(* Logix 5000 project; controller cal1632 1756-L62 rev 16.20; software revision 16.05; part 56 of 61 *)
(* tags used below, declared in another part *)
   abs_distance_to_move : REAL;   // Turret Absolute Distance to Move
   distance_to_move : REAL;   // Turret Distence to Move
   last_selected_position : REAL;   // Turret Last Selected Position
   p29_param_tension_hi_limit : REAL;   // Parameter Tension High Limit
   param_doff_position : REAL;
   param_pos_db : REAL;   // C: Turret Position Dead Band
   pb_jog_turret_rev : BOOL;   // HMI PB: Jog Turret Rev
   pos_hi_limit : REAL;   // Turret Position DB High Limit
   pos_hi_limit_temp : REAL;   // Turret Position High Limit Temp
   pos_lo_limit : REAL;   // Turret Position DB Low Limit
   pos_lo_limit_temp : REAL;   // Turret Position Low Limit Temp
   tmr_fwd_delay : TIMER;   // Turret Signal Dwell Timer
   tmr_ref_delay : TIMER;   // Turret Signal Dwell Timer
   turret_err_mod : REAL;   // Turret Shortest Path Error wrapped to 0..360
   turret_err_raw : REAL;   // Turret Shortest Path Raw error plus 540 offset
   turret_in_wda_run_position : BOOL;   // Turret In Winder A Run Position
   turret_in_wdb_run_position : BOOL;   // Turret In Winder B Run Position
   turret_index_active_last_scan : BOOL;   // Turret Index Active Last Scan
   turret_index_permissive : BOOL;   // Turret Index Permissive No Turret Drive Fault AND Neither Winder Requesting Run
   turret_request_reverse : BOOL;   // Turret Request Reverse Index
   turret_wa_pos_doff_request : BOOL;   // Turret Move to Winder A Doff Position Request
   turret_wa_pos_run_request : BOOL;   // Turret Move to Winder A Run Position
   turret_wb_pos_doff_request : BOOL;   // Turret Move to Winder B Doff Position Request
   turret_wb_pos_run_request : BOOL;   // Turret Move to Winder B Run Position
   wa_doff_pos : REAL;   // Turret Winder A Doff Position
   wb_doff_pos_tmp : REAL;   // Turret Temp Doff Position before MOD
   wb_doff_position : REAL;   // Turret Winder B Doff Position
   wb_run_position : REAL;   // Turret Winder B Run Position
   wb_run_position_tmp : REAL;   // Turret Temp Run Position before MOD
   FAULT : BOOL;
   HMI : BOOL;
   p01_param_tension_deviation : REAL;
   p01_recipe_active : recipe;
   p01r02_plc_scan_time_in_sec : REAL;
   p01r09_pb_global_reset : BOOL;
   p01r13_permissive_drives : BOOL;
   p01r13_state : DINT;
   p25_ao_selected_speed : REAL;
   p29_ai_wa_rpm : REAL;
   p29_ai_wb_rpm : REAL;
   p29_ai_wdr_dia_in : REAL;
   p29_ai_wdr_lc : REAL;
   p29_ao_wdr_turret_selected_speed : REAL;
   p29_di_wdr_a_core_size : BOOL;
   p29_di_wdr_a_reset_core : BOOL;
   p29_di_wdr_b_core_size : BOOL;
   p29_di_wdr_b_reset_core : BOOL;
   p29_di_wdr_index_fwd : BOOL;
   p29_di_wdr_turret : acs800_di_normal;
   p29_di_wt_motor : BOOL;
   p29_do_wdr_turret : acs800_do_normal;
   p29_param_fast_turret_speed : REAL;
   p29_param_slow_turret_speed : REAL;
   p29_param_wa_gear_ratio : REAL;
   p29_param_wb_gear_ratio : REAL;
   p29_winder_at_run_position : BOOL;
   p29r01 : routine;
   p29r09_mode_doff_auto : BOOL;   // Winder Mode Doff Position - AUTO Winder A/B doff PB indexes the turret to the preset doff position
   p29r09_ten_ave_len : DINT;
   p29r09_ten_len : DINT;
   p29r09_ten_pos : DINT;
   p29r09_torque_mode : BOOL;
   p29r09_trq_ave_len : DINT;
   p29r09_trq_len : DINT;
   p29r09_trq_pos : DINT;
   p29r10_pid_psn : PID;
   p29r11_pid_psn : PID;
   p29r15 : routine;
   p29r15_request_run : BOOL;
   p29r15_state : DINT;
   p29r15_wdra_active : BOOL;
   p29r16 : routine;
   p29r16_request_run : BOOL;
   p29r16_state : DINT;
   p29r16_wdrb_active : BOOL;
   p29r17 : routine;
   p29r17_ave_control : CONTROL;
   p29r17_diameter_clac_active : BOOL;
   p29r17_selected_core_diameter : REAL;
   p29r17_stack_ctrl : CONTROL;
   p29r17_timer : TIMER[5];
   p29r17_timer_fault : TIMER[4];
   p29r17_timer_warning : TIMER[4];
   p29r17_winder_a_actual_diam_inch : REAL;
   p29r17_winder_a_avg_diam_inch : REAL;
   p29r17_winder_a_calc_diam_inch : REAL;
   p29r17_winder_a_diam_avg_stack : REAL[1000];
   p29r17_winder_a_selected_diam_inch : REAL;
   p29r17_winder_a_unload : REAL;
   p29r18 : routine;
   p29r18_ave_control : CONTROL;
   p29r18_diameter_calc_active : BOOL;
   p29r18_min_tension : REAL;
   p29r18_selected_core_diameter : REAL;
   p29r18_stack_ctrl : CONTROL;
   p29r18_timer : TIMER[5];
   p29r18_timer_fault : TIMER[4];
   p29r18_timer_warning : TIMER[4];
   p29r18_winder_b_actual_diam_inch : REAL;
   p29r18_winder_b_avg_diam_inch : REAL;
   p29r18_winder_b_calc_diam_inch : REAL;
   p29r18_winder_b_diam_avg_stack : REAL[1000];
   p29r18_winder_b_selected_diam_inch : REAL;
   p29r18_winder_b_unload : REAL;
   p29r20 : routine;
   p29r20_acc_dec_ramp : SYS_ACC_DEC_RAMP;
   p29r20_accel_rate : REAL;
   p29r20_decel_rate : REAL;
   p29r20_fast_accel : REAL;
   p29r20_fast_decel : REAL;
   p29r20_index_complete : BOOL;
   p29r20_permissive : BOOL;
   p29r20_selected_speed : REAL;
   p29r20_timer_fault : TIMER[10];
   p29r20_timer_warning : TIMER[4];
   turret_in_position : BOOL;   // Turret In Position
(* P29_Winder, continued *)

ROUTINE R17_Winder_A_diameter_calc   (* ladder *)
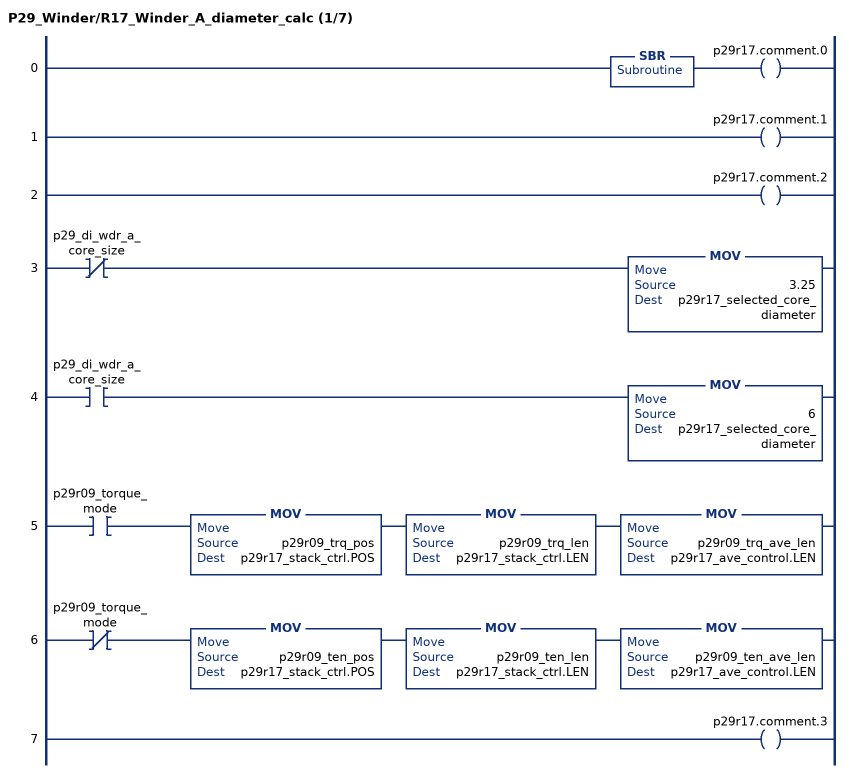
   0: SBR()OTE(p29r17.comment.0);
   1: OTE(p29r17.comment.1);
   2: OTE(p29r17.comment.2);
   3: XIO(p29_di_wdr_a_core_size)MOV(3.25,p29r17_selected_core_diameter);
   4: XIC(p29_di_wdr_a_core_size)MOV(6,p29r17_selected_core_diameter);
   5: XIC(p29r09_torque_mode)MOV(p29r09_trq_pos,p29r17_stack_ctrl.POS)MOV(p29r09_trq_len,p29r17_stack_ctrl.LEN)MOV(p29r09_trq_ave_len,p29r17_ave_control.LEN);
   6: XIO(p29r09_torque_mode)MOV(p29r09_ten_pos,p29r17_stack_ctrl.POS)MOV(p29r09_ten_len,p29r17_stack_ctrl.LEN)MOV(p29r09_ten_ave_len,p29r17_ave_control.LEN);
   7: OTE(p29r17.comment.3);
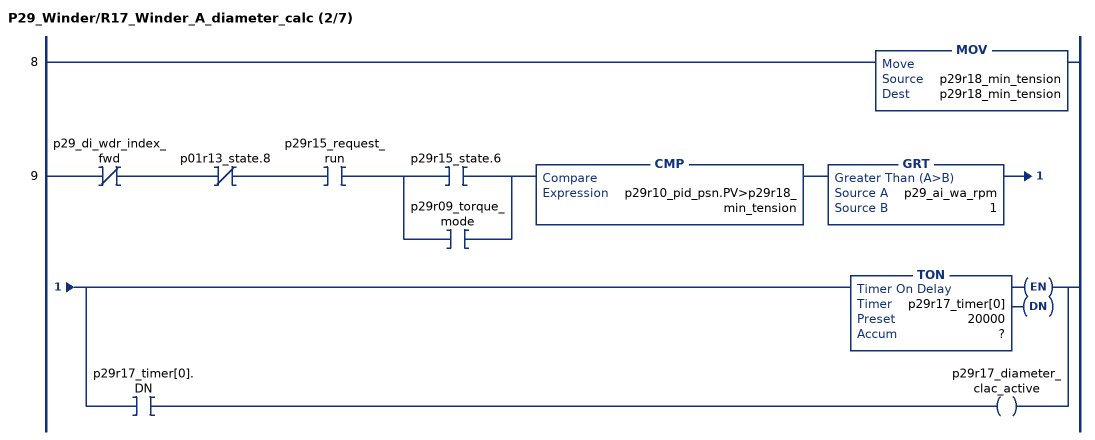
   8: MOV(p29r18_min_tension,p29r18_min_tension);
   9: XIO(p29_di_wdr_index_fwd)XIO(p01r13_state.8)XIC(p29r15_request_run)[XIC(p29r15_state.6) ,XIC(p29r09_torque_mode) ]CMP(p29r10_pid_psn.PV>p29r18_min_tension)GRT(p29_ai_wa_rpm,1)[TON(p29r17_timer[0],?,?) ,XIC(p29r17_timer[0].DN) OTE(p29r17_diameter_clac_active) ];
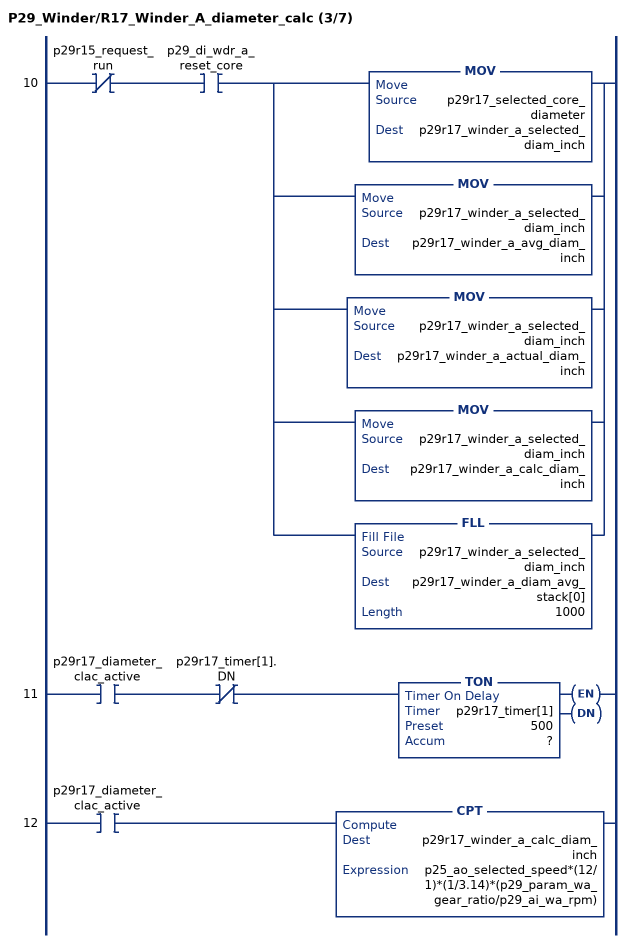
   10: XIO(p29r15_request_run)XIC(p29_di_wdr_a_reset_core)[MOV(p29r17_selected_core_diameter,p29r17_winder_a_selected_diam_inch) ,MOV(p29r17_winder_a_selected_diam_inch,p29r17_winder_a_avg_diam_inch) ,MOV(p29r17_winder_a_selected_diam_inch,p29r17_winder_a_actual_diam_inch) ,MOV(p29r17_winder_a_selected_diam_inch,p29r17_winder_a_calc_diam_inch) ,FLL(p29r17_winder_a_selected_diam_inch,p29r17_winder_a_diam_avg_stack[0],1000) ];
   11: XIC(p29r17_diameter_clac_active)XIO(p29r17_timer[1].DN)TON(p29r17_timer[1],?,?);
   12: XIC(p29r17_diameter_clac_active)CPT(p29r17_winder_a_calc_diam_inch,p25_ao_selected_speed*(12/1)*(1/3.14)*(p29_param_wa_gear_ratio/p29_ai_wa_rpm));
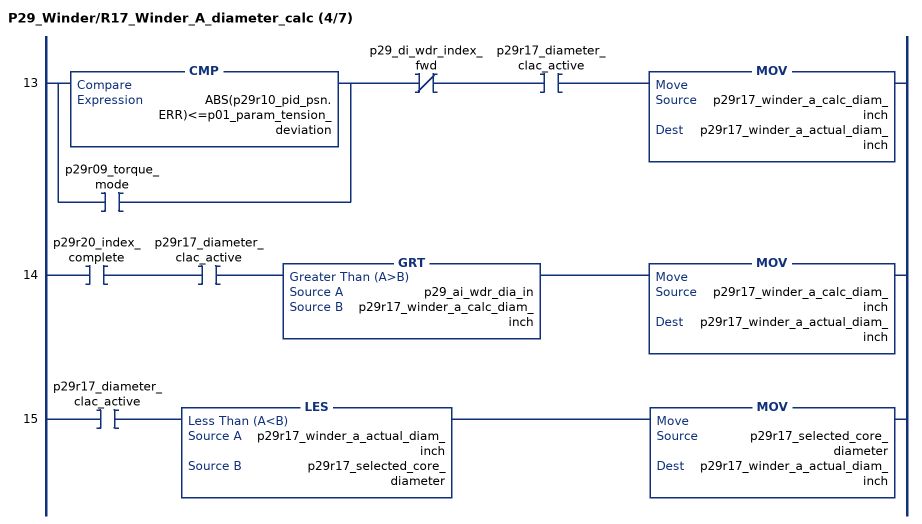
   13: [CMP(ABS(p29r10_pid_psn.ERR)<=p01_param_tension_deviation) ,XIC(p29r09_torque_mode) ]XIO(p29_di_wdr_index_fwd)XIC(p29r17_diameter_clac_active)MOV(p29r17_winder_a_calc_diam_inch,p29r17_winder_a_actual_diam_inch);
   14: XIC(p29r20_index_complete)XIC(p29r17_diameter_clac_active)GRT(p29_ai_wdr_dia_in,p29r17_winder_a_calc_diam_inch)MOV(p29r17_winder_a_calc_diam_inch,p29r17_winder_a_actual_diam_inch);
   15: XIC(p29r17_diameter_clac_active)LES(p29r17_winder_a_actual_diam_inch,p29r17_selected_core_diameter)MOV(p29r17_selected_core_diameter,p29r17_winder_a_actual_diam_inch);
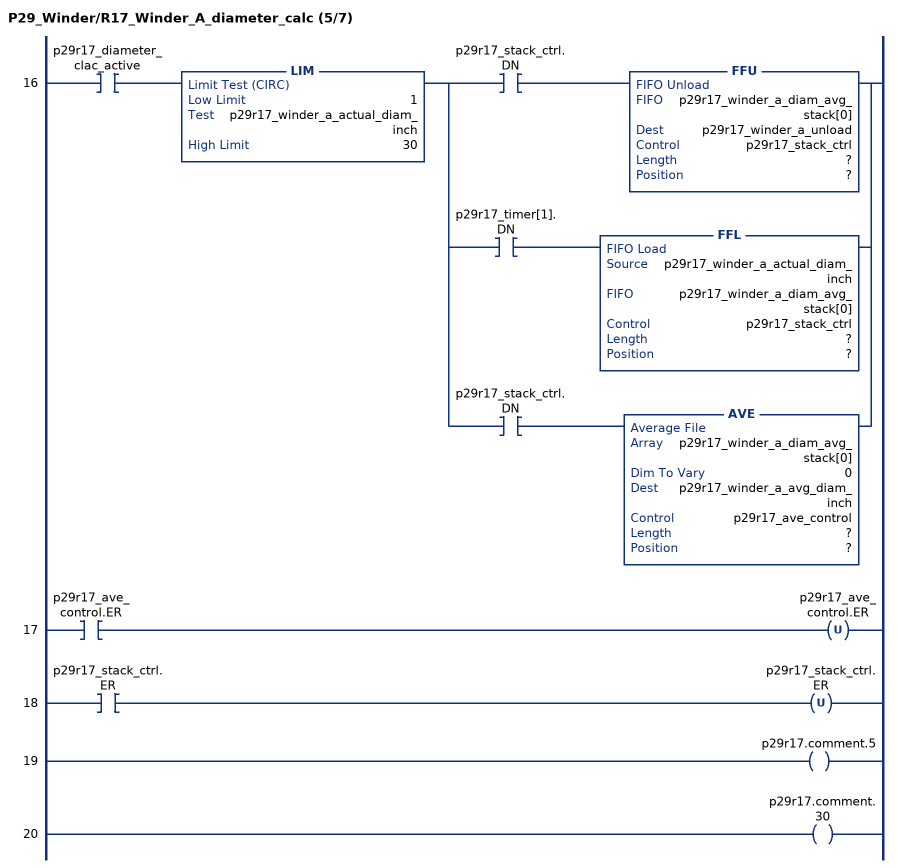
   16: XIC(p29r17_diameter_clac_active)LIM(1,p29r17_winder_a_actual_diam_inch,30)[XIC(p29r17_stack_ctrl.DN) FFU(p29r17_winder_a_diam_avg_stack[0],p29r17_winder_a_unload,p29r17_stack_ctrl,?,?) ,XIC(p29r17_timer[1].DN) FFL(p29r17_winder_a_actual_diam_inch,p29r17_winder_a_diam_avg_stack[0],p29r17_stack_ctrl,?,?) ,XIC(p29r17_stack_ctrl.DN) AVE(p29r17_winder_a_diam_avg_stack[0],0,p29r17_winder_a_avg_diam_inch,p29r17_ave_control,?,?) ];
   17: XIC(p29r17_ave_control.ER)OTU(p29r17_ave_control.ER);
   18: XIC(p29r17_stack_ctrl.ER)OTU(p29r17_stack_ctrl.ER);
   19: OTE(p29r17.comment.5);
   20: OTE(p29r17.comment.30);
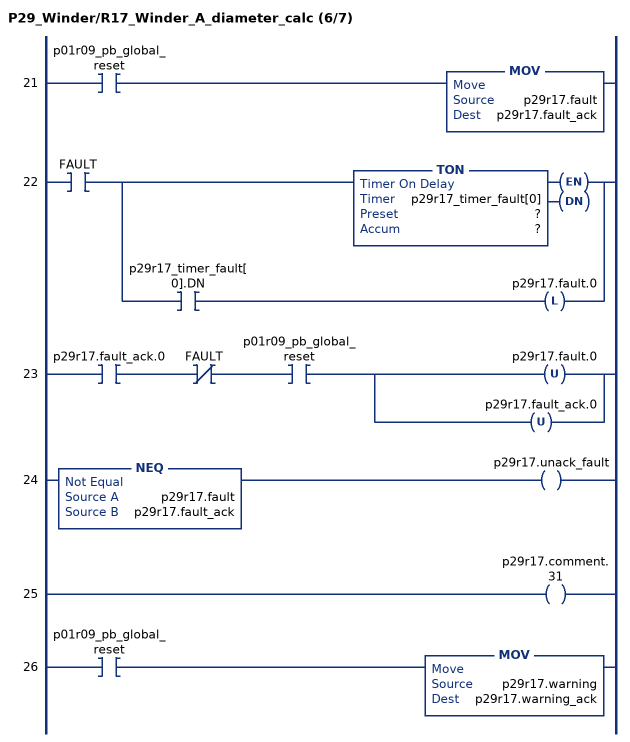
   21: XIC(p01r09_pb_global_reset)MOV(p29r17.fault,p29r17.fault_ack);
   22: XIC(FAULT)[TON(p29r17_timer_fault[0],?,?) ,XIC(p29r17_timer_fault[0].DN) OTL(p29r17.fault.0) ];
   23: XIC(p29r17.fault_ack.0)XIO(FAULT)XIC(p01r09_pb_global_reset)[OTU(p29r17.fault.0) ,OTU(p29r17.fault_ack.0) ];
   24: NEQ(p29r17.fault,p29r17.fault_ack)OTE(p29r17.unack_fault);
   25: OTE(p29r17.comment.31);
   26: XIC(p01r09_pb_global_reset)MOV(p29r17.warning,p29r17.warning_ack);
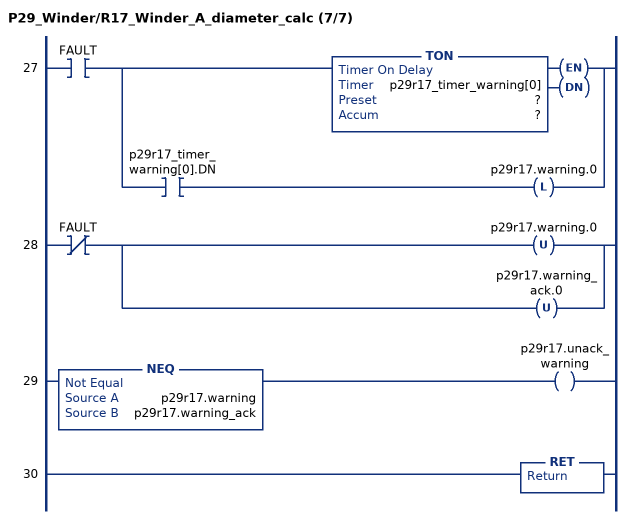
   27: XIC(FAULT)[TON(p29r17_timer_warning[0],?,?) ,XIC(p29r17_timer_warning[0].DN) OTL(p29r17.warning.0) ];
   28: XIO(FAULT)[OTU(p29r17.warning.0) ,OTU(p29r17.warning_ack.0) ];
   29: NEQ(p29r17.warning,p29r17.warning_ack)OTE(p29r17.unack_warning);
   30: RET();
END_ROUTINE

ROUTINE R18_Winder_B_diameter_calc   (* ladder *)
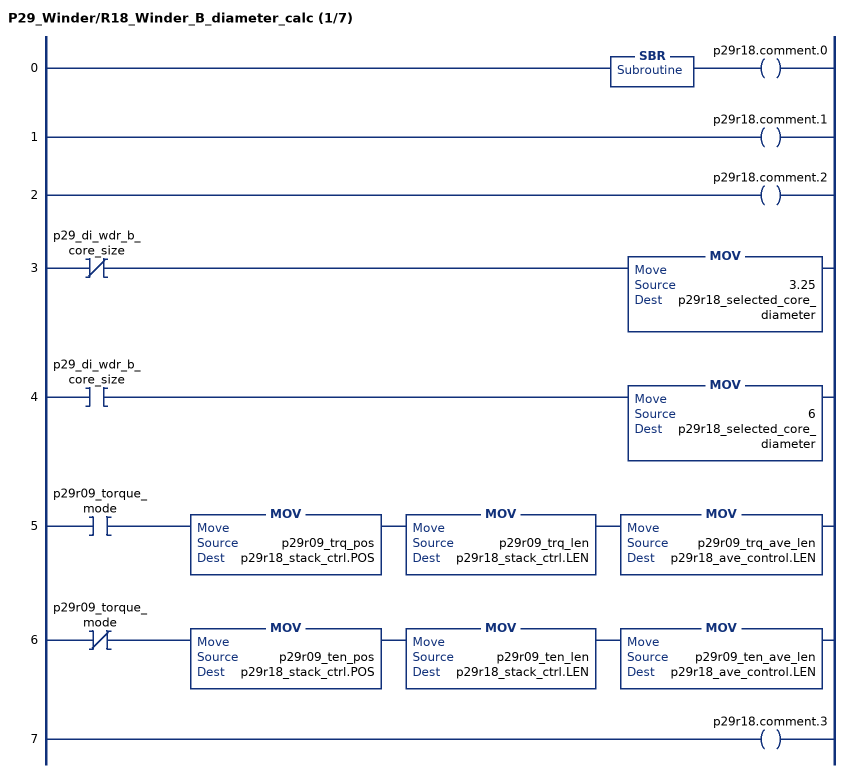
   0: SBR()OTE(p29r18.comment.0);
   1: OTE(p29r18.comment.1);
   2: OTE(p29r18.comment.2);
   3: XIO(p29_di_wdr_b_core_size)MOV(3.25,p29r18_selected_core_diameter);
   4: XIC(p29_di_wdr_b_core_size)MOV(6,p29r18_selected_core_diameter);
   5: XIC(p29r09_torque_mode)MOV(p29r09_trq_pos,p29r18_stack_ctrl.POS)MOV(p29r09_trq_len,p29r18_stack_ctrl.LEN)MOV(p29r09_trq_ave_len,p29r18_ave_control.LEN);
   6: XIO(p29r09_torque_mode)MOV(p29r09_ten_pos,p29r18_stack_ctrl.POS)MOV(p29r09_ten_len,p29r18_stack_ctrl.LEN)MOV(p29r09_ten_ave_len,p29r18_ave_control.LEN);
   7: OTE(p29r18.comment.3);
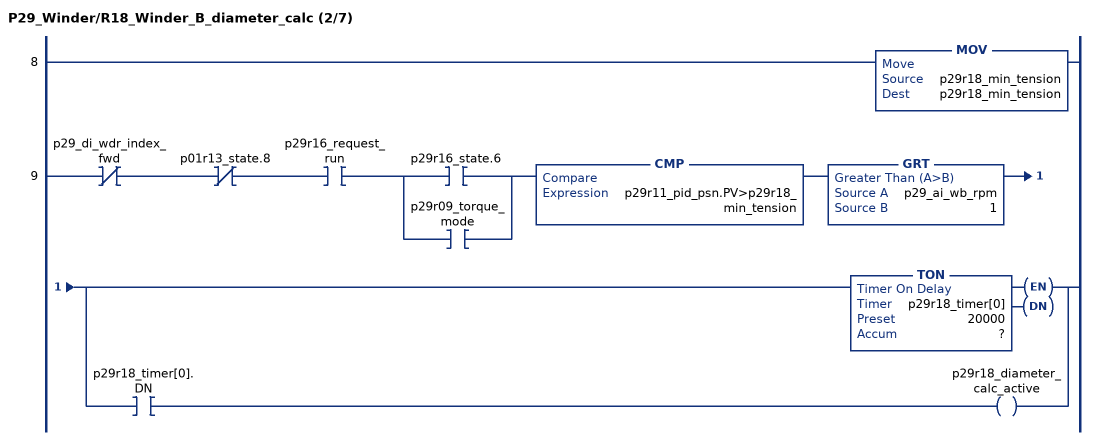
   8: MOV(p29r18_min_tension,p29r18_min_tension);
   9: XIO(p29_di_wdr_index_fwd)XIO(p01r13_state.8)XIC(p29r16_request_run)[XIC(p29r16_state.6) ,XIC(p29r09_torque_mode) ]CMP(p29r11_pid_psn.PV>p29r18_min_tension)GRT(p29_ai_wb_rpm,1)[TON(p29r18_timer[0],?,?) ,XIC(p29r18_timer[0].DN) OTE(p29r18_diameter_calc_active) ];
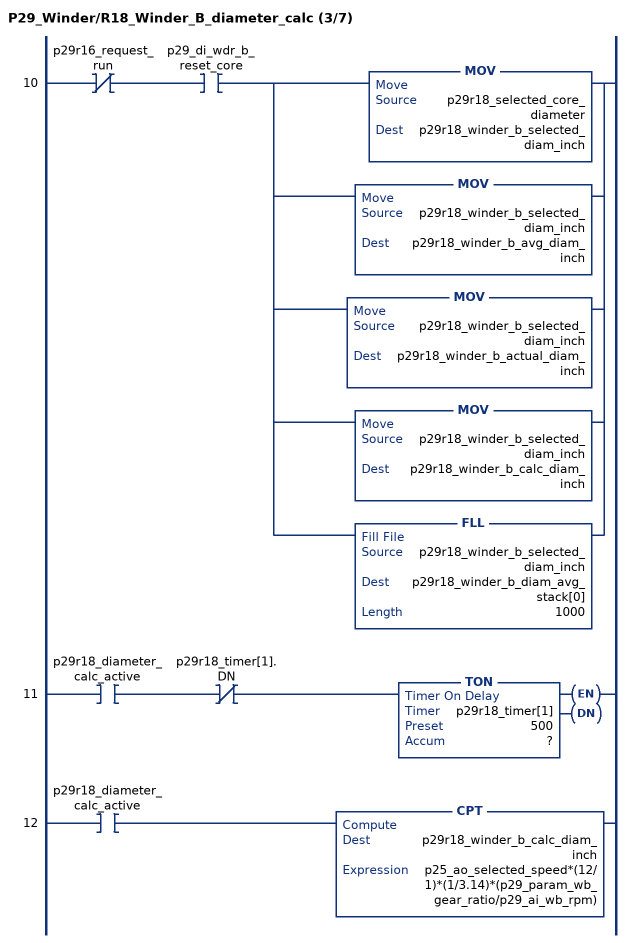
   10: XIO(p29r16_request_run)XIC(p29_di_wdr_b_reset_core)[MOV(p29r18_selected_core_diameter,p29r18_winder_b_selected_diam_inch) ,MOV(p29r18_winder_b_selected_diam_inch,p29r18_winder_b_avg_diam_inch) ,MOV(p29r18_winder_b_selected_diam_inch,p29r18_winder_b_actual_diam_inch) ,MOV(p29r18_winder_b_selected_diam_inch,p29r18_winder_b_calc_diam_inch) ,FLL(p29r18_winder_b_selected_diam_inch,p29r18_winder_b_diam_avg_stack[0],1000) ];
   11: XIC(p29r18_diameter_calc_active)XIO(p29r18_timer[1].DN)TON(p29r18_timer[1],?,?);
   12: XIC(p29r18_diameter_calc_active)CPT(p29r18_winder_b_calc_diam_inch,p25_ao_selected_speed*(12/1)*(1/3.14)*(p29_param_wb_gear_ratio/p29_ai_wb_rpm));
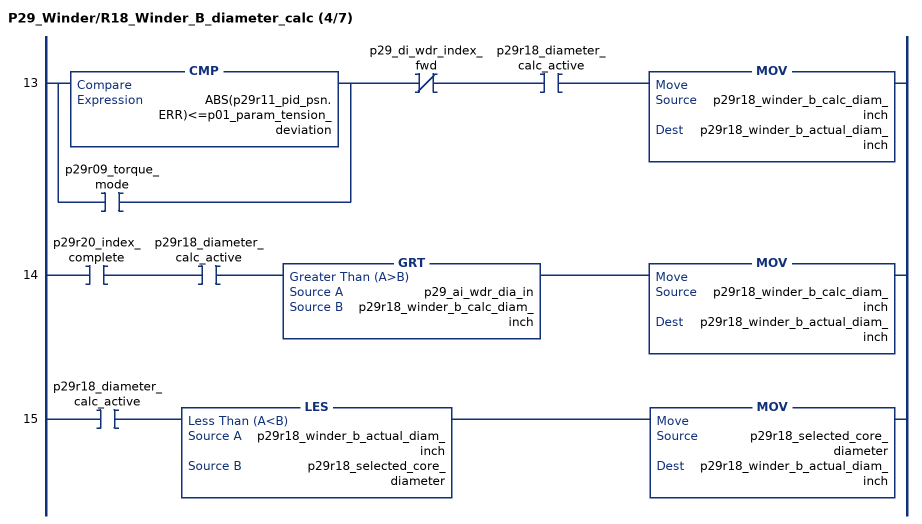
   13: [CMP(ABS(p29r11_pid_psn.ERR)<=p01_param_tension_deviation) ,XIC(p29r09_torque_mode) ]XIO(p29_di_wdr_index_fwd)XIC(p29r18_diameter_calc_active)MOV(p29r18_winder_b_calc_diam_inch,p29r18_winder_b_actual_diam_inch);
   14: XIC(p29r20_index_complete)XIC(p29r18_diameter_calc_active)GRT(p29_ai_wdr_dia_in,p29r18_winder_b_calc_diam_inch)MOV(p29r18_winder_b_calc_diam_inch,p29r18_winder_b_actual_diam_inch);
   15: XIC(p29r18_diameter_calc_active)LES(p29r18_winder_b_actual_diam_inch,p29r18_selected_core_diameter)MOV(p29r18_selected_core_diameter,p29r18_winder_b_actual_diam_inch);
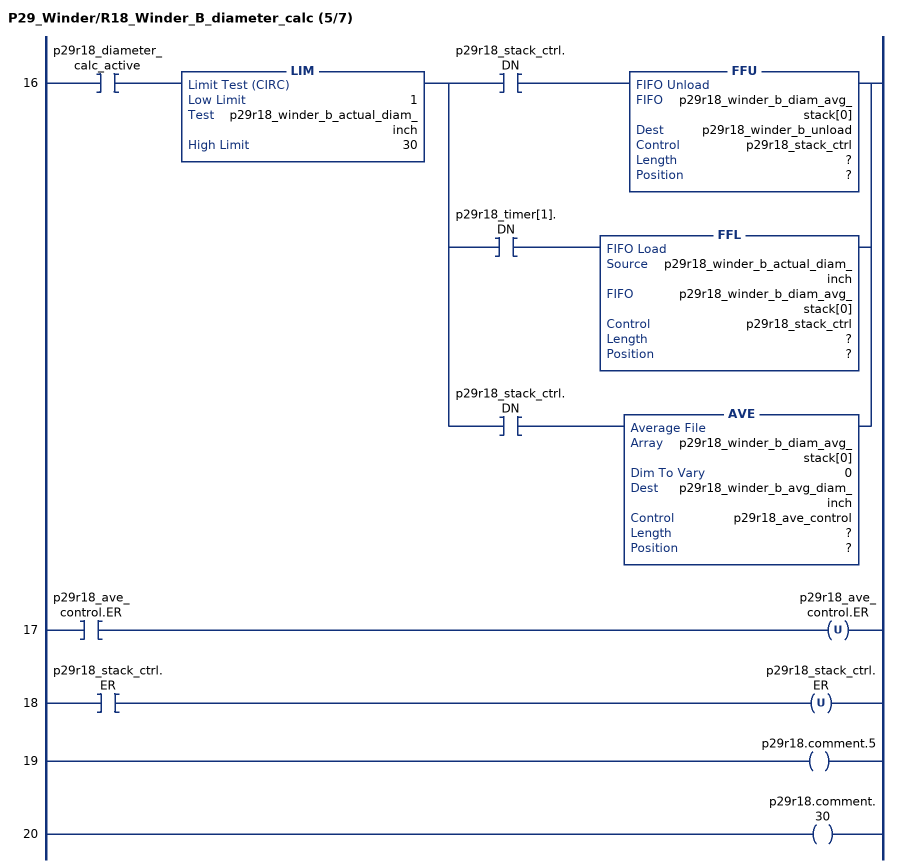
   16: XIC(p29r18_diameter_calc_active)LIM(1,p29r18_winder_b_actual_diam_inch,30)[XIC(p29r18_stack_ctrl.DN) FFU(p29r18_winder_b_diam_avg_stack[0],p29r18_winder_b_unload,p29r18_stack_ctrl,?,?) ,XIC(p29r18_timer[1].DN) FFL(p29r18_winder_b_actual_diam_inch,p29r18_winder_b_diam_avg_stack[0],p29r18_stack_ctrl,?,?) ,XIC(p29r18_stack_ctrl.DN) AVE(p29r18_winder_b_diam_avg_stack[0],0,p29r18_winder_b_avg_diam_inch,p29r18_ave_control,?,?) ];
   17: XIC(p29r18_ave_control.ER)OTU(p29r18_ave_control.ER);
   18: XIC(p29r18_stack_ctrl.ER)OTU(p29r18_stack_ctrl.ER);
   19: OTE(p29r18.comment.5);
   20: OTE(p29r18.comment.30);
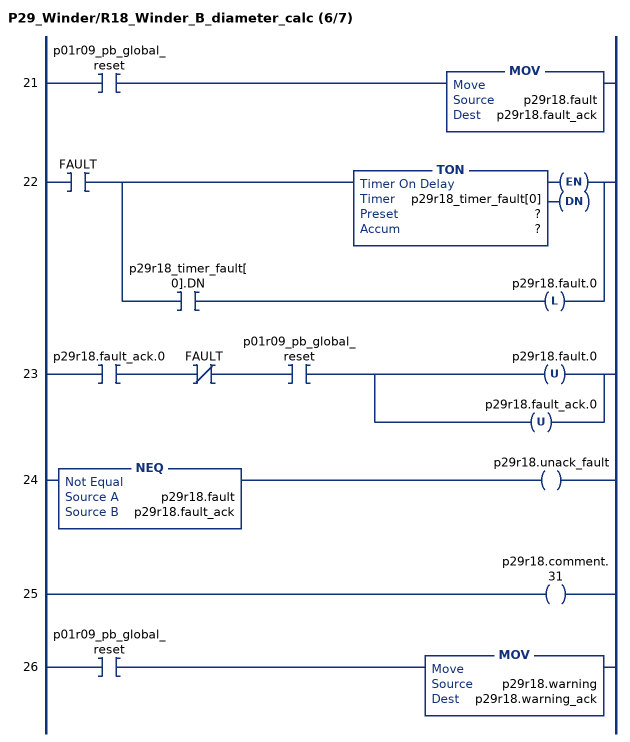
   21: XIC(p01r09_pb_global_reset)MOV(p29r18.fault,p29r18.fault_ack);
   22: XIC(FAULT)[TON(p29r18_timer_fault[0],?,?) ,XIC(p29r18_timer_fault[0].DN) OTL(p29r18.fault.0) ];
   23: XIC(p29r18.fault_ack.0)XIO(FAULT)XIC(p01r09_pb_global_reset)[OTU(p29r18.fault.0) ,OTU(p29r18.fault_ack.0) ];
   24: NEQ(p29r18.fault,p29r18.fault_ack)OTE(p29r18.unack_fault);
   25: OTE(p29r18.comment.31);
   26: XIC(p01r09_pb_global_reset)MOV(p29r18.warning,p29r18.warning_ack);
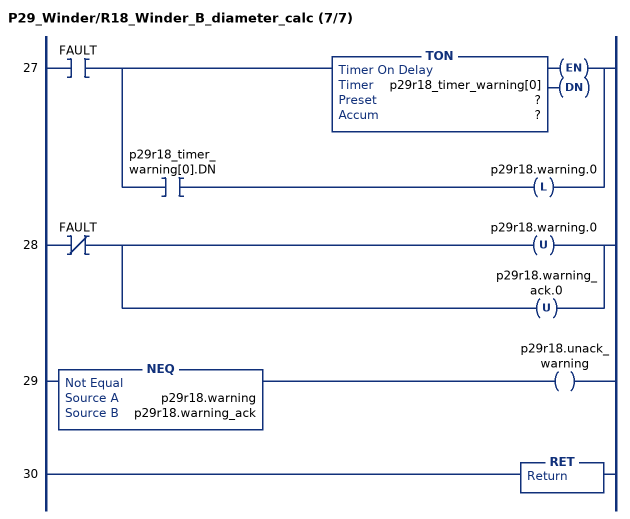
   27: XIC(FAULT)[TON(p29r18_timer_warning[0],?,?) ,XIC(p29r18_timer_warning[0].DN) OTL(p29r18.warning.0) ];
   28: XIO(FAULT)[OTU(p29r18.warning.0) ,OTU(p29r18.warning_ack.0) ];
   29: NEQ(p29r18.warning,p29r18.warning_ack)OTE(p29r18.unack_warning);
   30: RET();
END_ROUTINE

ROUTINE R20_Winder_Turret_VFD   (* ladder *)
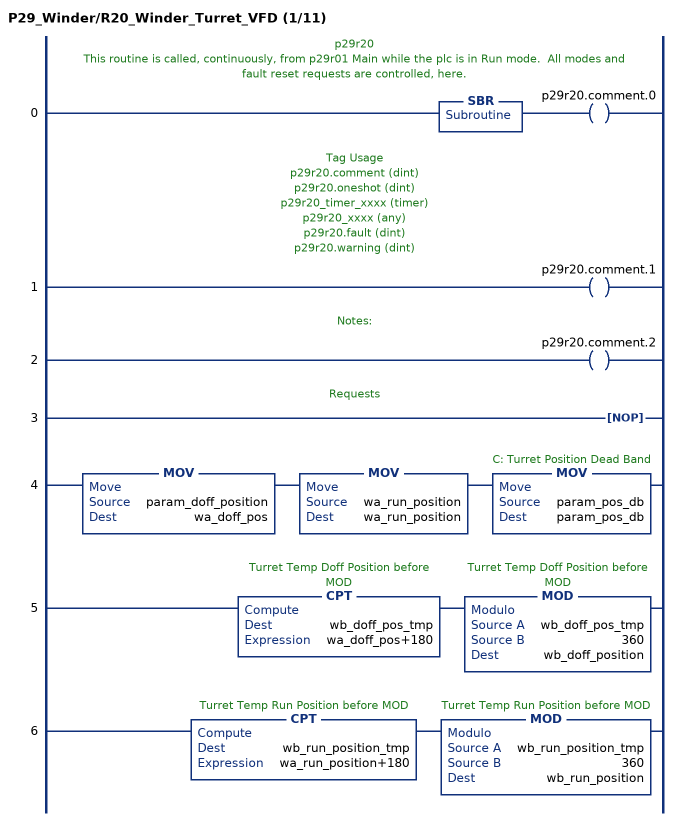
   // p29r20
   // This routine is called, continuously, from p29r01 Main while the plc is in Run mode.  All modes and fault reset requests are controlled, here.
   0: SBR()OTE(p29r20.comment.0);
   // Tag Usage
   // p29r20.comment (dint)
   // p29r20.oneshot (dint)
   // p29r20_timer_xxxx (timer)
   // p29r20_xxxx (any)
   // p29r20.fault (dint)
   // p29r20.warning (dint)
   1: OTE(p29r20.comment.1);
   // Notes:
   2: OTE(p29r20.comment.2);
   // Requests
   3: NOP();
   4: MOV(param_doff_position,wa_doff_pos)MOV(wa_run_position,wa_run_position)MOV(param_pos_db,param_pos_db);
   5: CPT(wb_doff_pos_tmp,wa_doff_pos+180)MOD(wb_doff_pos_tmp,360,wb_doff_position);
   6: CPT(wb_run_position_tmp,wa_run_position+180)MOD(wb_run_position_tmp,360,wb_run_position);
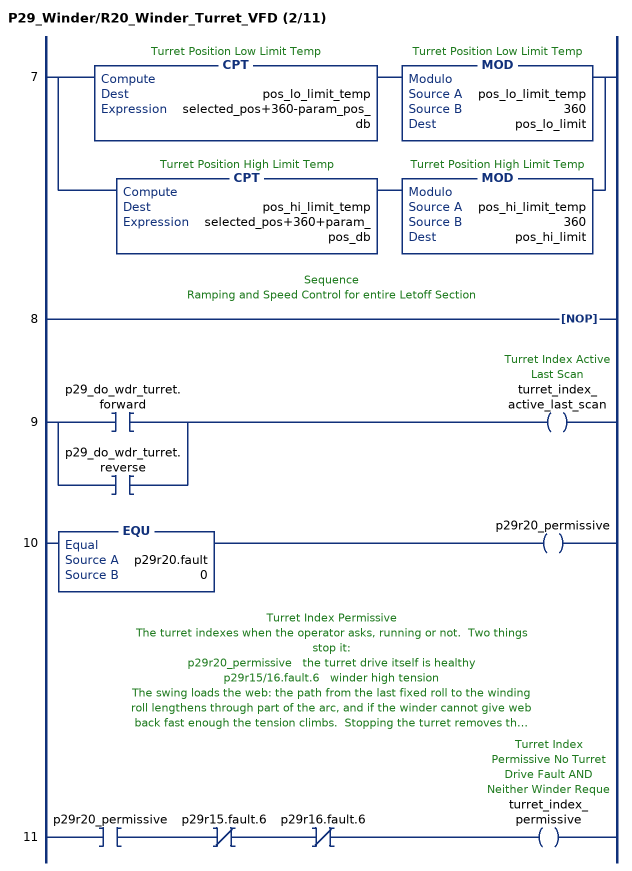
   7: [CPT(pos_lo_limit_temp,selected_pos+360-param_pos_db) MOD(pos_lo_limit_temp,360,pos_lo_limit) ,CPT(pos_hi_limit_temp,selected_pos+360+param_pos_db) MOD(pos_hi_limit_temp,360,pos_hi_limit) ];
   // Sequence
   // Ramping and Speed Control for entire Letoff Section
   8: NOP();
   9: [XIC(p29_do_wdr_turret.forward) ,XIC(p29_do_wdr_turret.reverse) ]OTE(turret_index_active_last_scan);
   10: EQU(p29r20.fault,0)OTE(p29r20_permissive);
   // Turret Index Permissive
   // The turret indexes when the operator asks, running or not.  Two things
   // stop it:
   //   p29r20_permissive   the turret drive itself is healthy
   //   p29r15/16.fault.6   winder high tension
   // The swing loads the web: the path from the last fixed roll to the winding
   // roll lengthens through part of the arc, and if the winder cannot give web
   // back fast enough the tension climbs.  Stopping the turret removes the
   // cause; carrying on pulls against it.
   // Both winders are tested, not just the selected one.  fault.6 latches until
   // a global reset, so a stale fault on the idle winder will hold the turret
   // until it is acknowledged - deliberate.
   // fault.6 = GRT(p29_ai_wdr_lc, p29_param_tension_hi_limit), 20 lbf
   // hysteresis on the reset.
   // Rev 20260825 a31
   11: XIC(p29r20_permissive)XIO(p29r15.fault.6)XIO(p29r16.fault.6)OTE(turret_index_permissive);
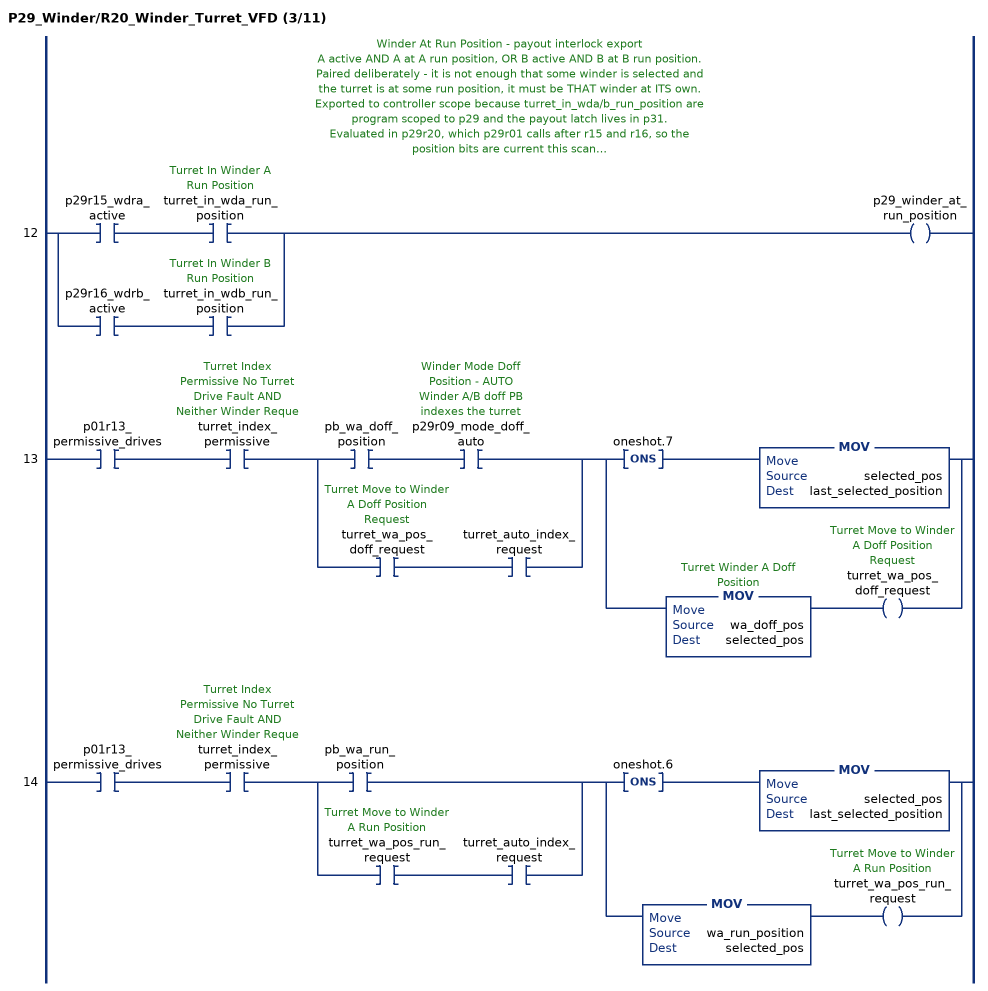
   // Winder At Run Position - payout interlock export
   // A active AND A at A run position, OR B active AND B at B run position.
   // Paired deliberately - it is not enough that some winder is selected and
   // the turret is at some run position, it must be THAT winder at ITS own.
   // Exported to controller scope because turret_in_wda/b_run_position are
   // program scoped to p29 and the payout latch lives in p31.
   // Evaluated in p29r20, which p29r01 calls after r15 and r16, so the
   // position bits are current this scan.
   // Rev 20260829 a33
   12: [XIC(p29r15_wdra_active) XIC(turret_in_wda_run_position) ,XIC(p29r16_wdrb_active) XIC(turret_in_wdb_run_position) ]OTE(p29_winder_at_run_position);
   13: XIC(p01r13_permissive_drives)XIC(turret_index_permissive)[XIC(pb_wa_doff_position) XIC(p29r09_mode_doff_auto) ,XIC(turret_wa_pos_doff_request) XIC(turret_auto_index_request) ][ONS(oneshot.7) MOV(selected_pos,last_selected_position) ,MOV(wa_doff_pos,selected_pos) OTE(turret_wa_pos_doff_request) ];
   14: XIC(p01r13_permissive_drives)XIC(turret_index_permissive)[XIC(pb_wa_run_position) ,XIC(turret_wa_pos_run_request) XIC(turret_auto_index_request) ][ONS(oneshot.6) MOV(selected_pos,last_selected_position) ,MOV(wa_run_position,selected_pos) OTE(turret_wa_pos_run_request) ];
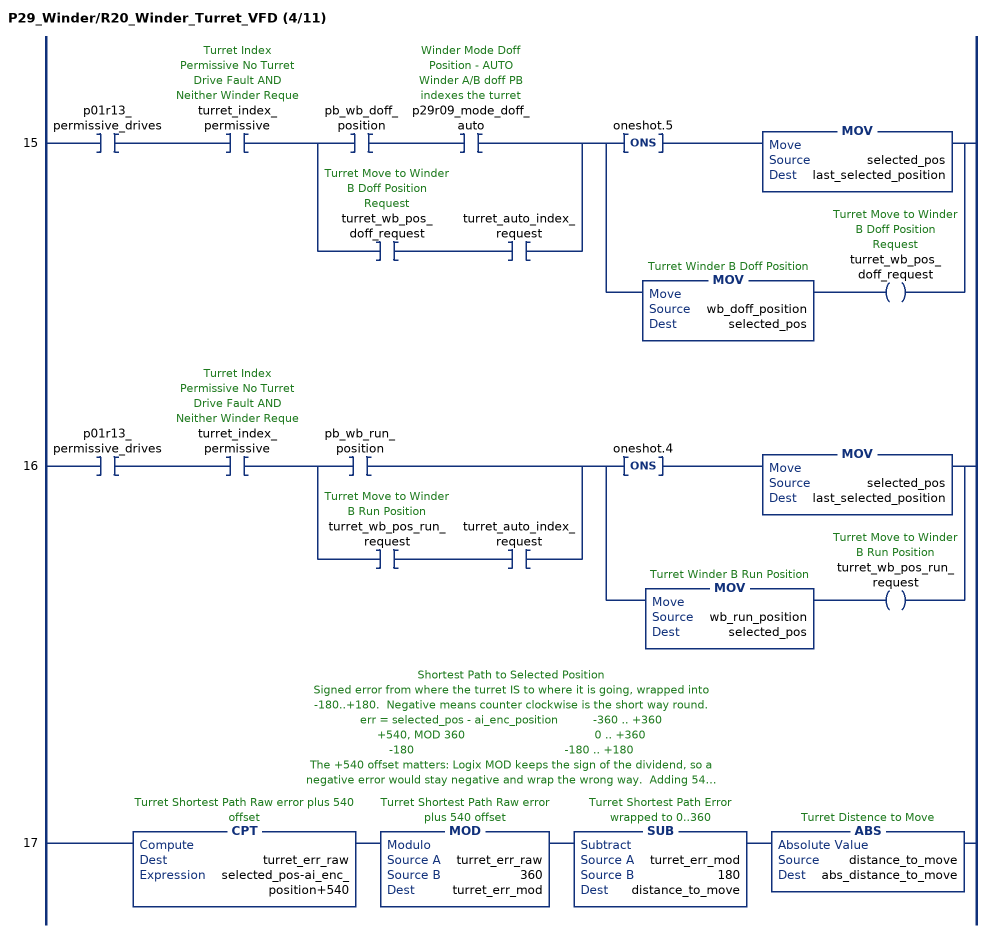
   15: XIC(p01r13_permissive_drives)XIC(turret_index_permissive)[XIC(pb_wb_doff_position) XIC(p29r09_mode_doff_auto) ,XIC(turret_wb_pos_doff_request) XIC(turret_auto_index_request) ][ONS(oneshot.5) MOV(selected_pos,last_selected_position) ,MOV(wb_doff_position,selected_pos) OTE(turret_wb_pos_doff_request) ];
   16: XIC(p01r13_permissive_drives)XIC(turret_index_permissive)[XIC(pb_wb_run_position) ,XIC(turret_wb_pos_run_request) XIC(turret_auto_index_request) ][ONS(oneshot.4) MOV(selected_pos,last_selected_position) ,MOV(wb_run_position,selected_pos) OTE(turret_wb_pos_run_request) ];
   // Shortest Path to Selected Position
   // Signed error from where the turret IS to where it is going, wrapped into
   // -180..+180.  Negative means counter clockwise is the short way round.
   //   err = selected_pos - ai_enc_position          -360 .. +360
   //   +540, MOD 360                                     0 .. +360
   //   -180                                           -180 .. +180
   // The +540 offset matters: Logix MOD keeps the sign of the dividend, so a
   // negative error would stay negative and wrap the wrong way.  Adding 540
   // puts the argument in 180..900, always positive, before the MOD.
   // Evaluated continuously, not one shot on the request.  The old rung took
   // SUB(last_selected_position, selected_pos) - the distance between the two
   // most recent TARGETS, not the distance from where the turret actually is.
   // After a jog, or an aborted index, that is simply the wrong number.  Live
   // evaluation also corrects an overshoot instead of driving on round.
   // Replaces the old 45 deg threshold test and the mode_under HMI override,
   // which picked direction by rules rather than by which way was shorter.
   // A run and B run are 180 deg apart, so a run-to-run move is exactly
   // antipodal and resolves to reverse.  Deterministic, but if that is the
   // wrong way round the machine, bias one run position by a degree.
   // Rev 20260825 a25
   17: CPT(turret_err_raw,selected_pos-ai_enc_position+540)MOD(turret_err_raw,360,turret_err_mod)SUB(turret_err_mod,180,distance_to_move)ABS(distance_to_move,abs_distance_to_move);
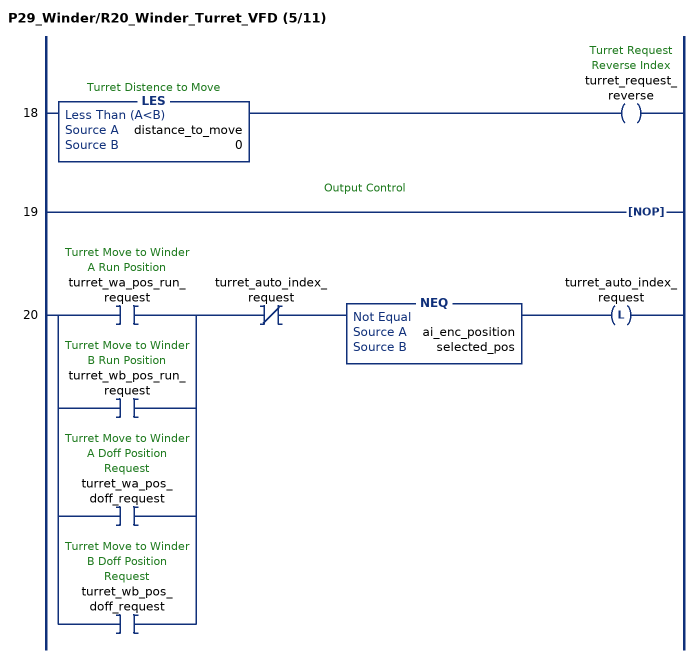
   18: LES(distance_to_move,0)OTE(turret_request_reverse);
   // Output Control
   19: NOP();
   20: [XIC(turret_wa_pos_run_request) ,XIC(turret_wb_pos_run_request) ,XIC(turret_wa_pos_doff_request) ,XIC(turret_wb_pos_doff_request) ]XIO(turret_auto_index_request)NEQ(ai_enc_position,selected_pos)OTL(turret_auto_index_request);
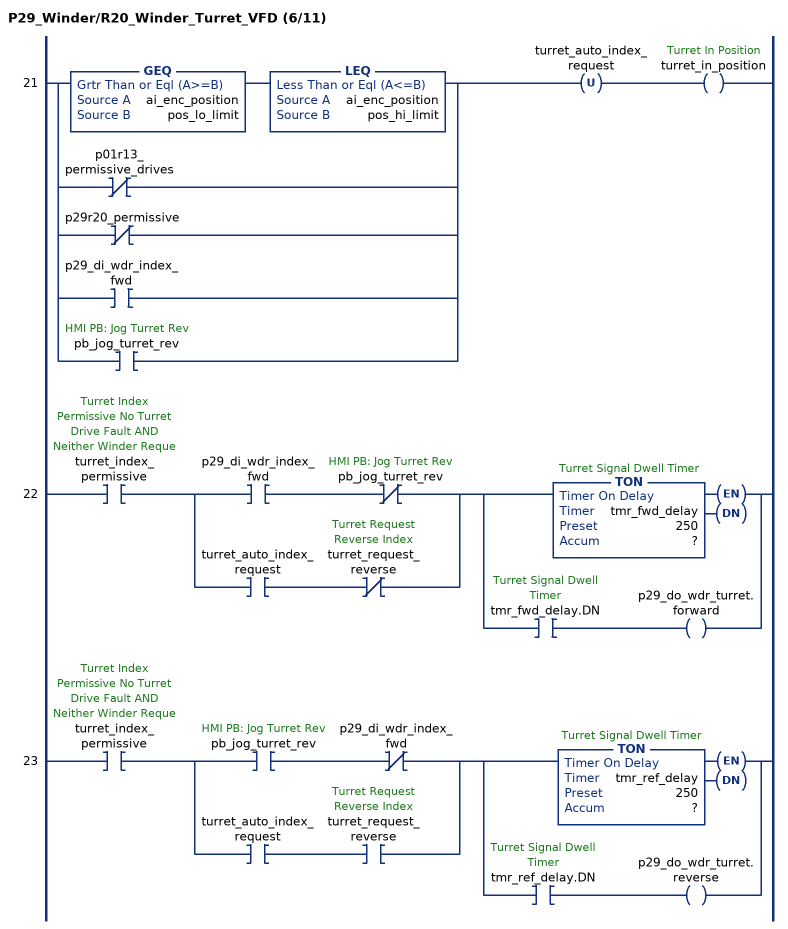
   21: [GEQ(ai_enc_position,pos_lo_limit) LEQ(ai_enc_position,pos_hi_limit) ,XIO(p01r13_permissive_drives) ,XIO(p29r20_permissive) ,XIC(p29_di_wdr_index_fwd) ,XIC(pb_jog_turret_rev) ]OTU(turret_auto_index_request)OTE(turret_in_position);
   22: XIC(turret_index_permissive)[XIC(p29_di_wdr_index_fwd) XIO(pb_jog_turret_rev) ,XIC(turret_auto_index_request) XIO(turret_request_reverse) ][TON(tmr_fwd_delay,?,?) ,XIC(tmr_fwd_delay.DN) OTE(p29_do_wdr_turret.forward) ];
   23: XIC(turret_index_permissive)[XIC(pb_jog_turret_rev) XIO(p29_di_wdr_index_fwd) ,XIC(turret_auto_index_request) XIC(turret_request_reverse) ][TON(tmr_ref_delay,?,?) ,XIC(tmr_ref_delay.DN) OTE(p29_do_wdr_turret.reverse) ];
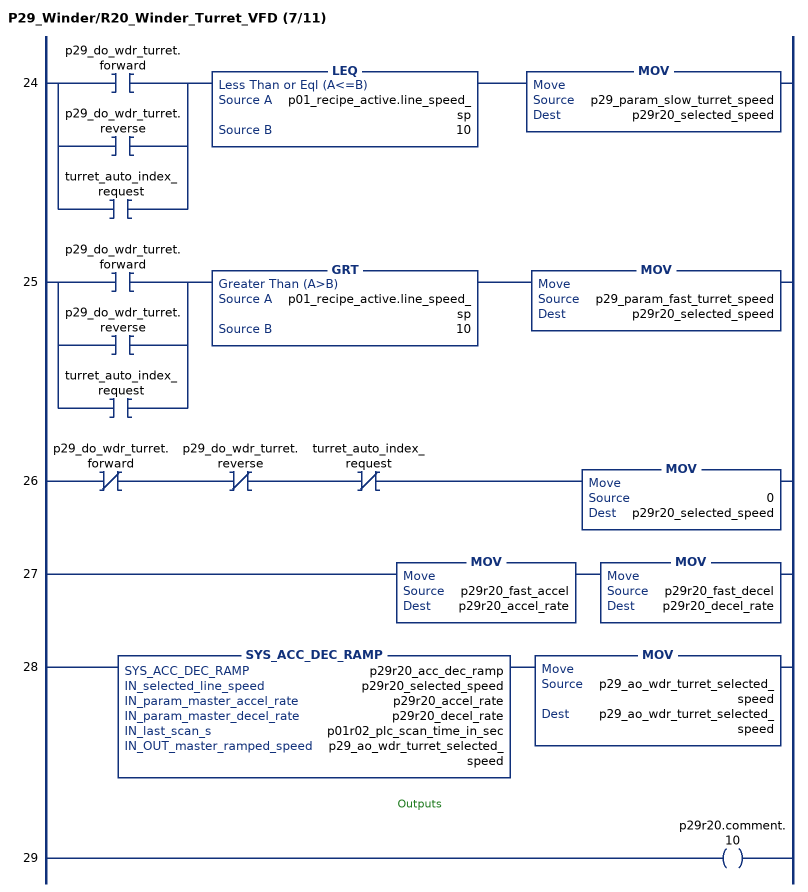
   24: [XIC(p29_do_wdr_turret.forward) ,XIC(p29_do_wdr_turret.reverse) ,XIC(turret_auto_index_request) ]LEQ(p01_recipe_active.line_speed_sp,10)MOV(p29_param_slow_turret_speed,p29r20_selected_speed);
   25: [XIC(p29_do_wdr_turret.forward) ,XIC(p29_do_wdr_turret.reverse) ,XIC(turret_auto_index_request) ]GRT(p01_recipe_active.line_speed_sp,10)MOV(p29_param_fast_turret_speed,p29r20_selected_speed);
   26: XIO(p29_do_wdr_turret.forward)XIO(p29_do_wdr_turret.reverse)XIO(turret_auto_index_request)MOV(0,p29r20_selected_speed);
   27: MOV(p29r20_fast_accel,p29r20_accel_rate)MOV(p29r20_fast_decel,p29r20_decel_rate);
   28: SYS_ACC_DEC_RAMP(p29r20_acc_dec_ramp,p29r20_selected_speed,p29r20_accel_rate,p29r20_decel_rate,p01r02_plc_scan_time_in_sec,p29_ao_wdr_turret_selected_speed)MOV(p29_ao_wdr_turret_selected_speed,p29_ao_wdr_turret_selected_speed);
   // Outputs
   29: OTE(p29r20.comment.10);
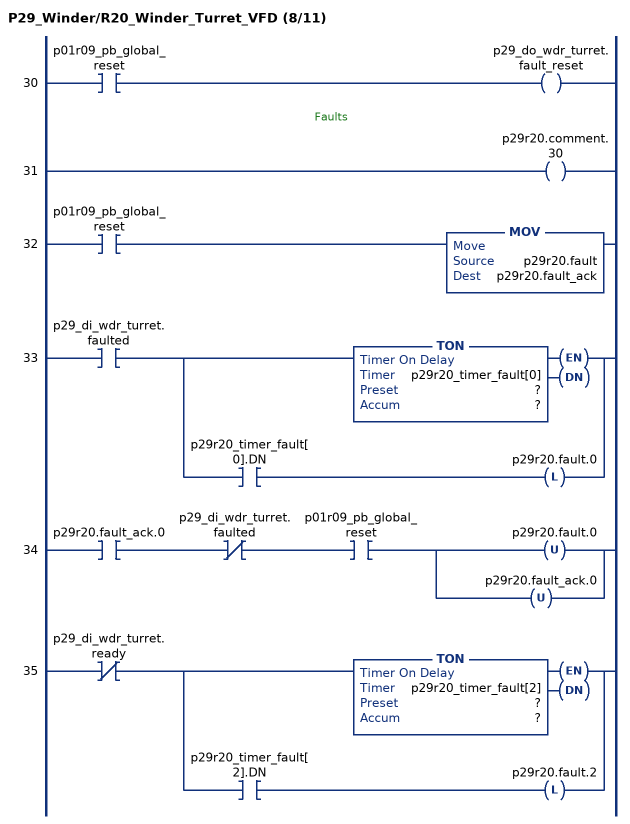
   30: XIC(p01r09_pb_global_reset)OTE(p29_do_wdr_turret.fault_reset);
   // Faults
   31: OTE(p29r20.comment.30);
   32: XIC(p01r09_pb_global_reset)MOV(p29r20.fault,p29r20.fault_ack);
   33: XIC(p29_di_wdr_turret.faulted)[TON(p29r20_timer_fault[0],?,?) ,XIC(p29r20_timer_fault[0].DN) OTL(p29r20.fault.0) ];
   34: XIC(p29r20.fault_ack.0)XIO(p29_di_wdr_turret.faulted)XIC(p01r09_pb_global_reset)[OTU(p29r20.fault.0) ,OTU(p29r20.fault_ack.0) ];
   35: XIO(p29_di_wdr_turret.ready)[TON(p29r20_timer_fault[2],?,?) ,XIC(p29r20_timer_fault[2].DN) OTL(p29r20.fault.2) ];
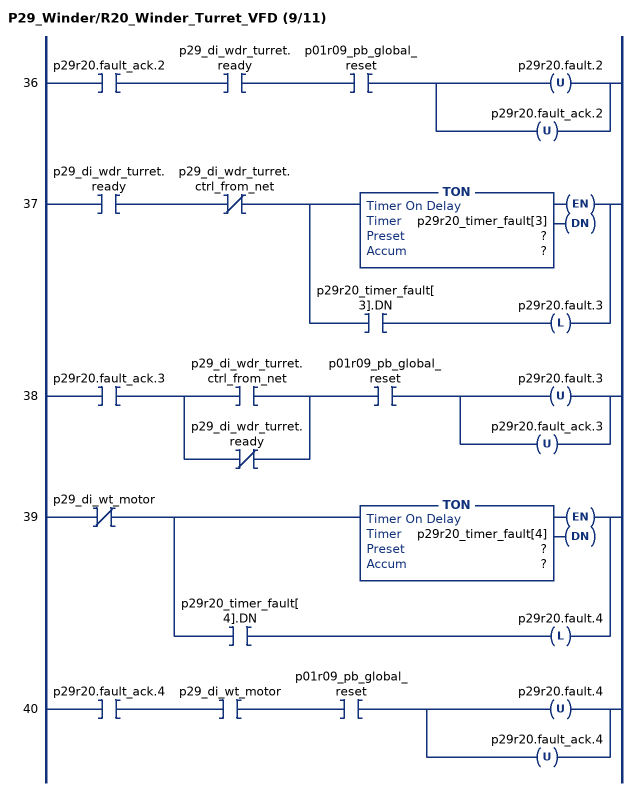
   36: XIC(p29r20.fault_ack.2)XIC(p29_di_wdr_turret.ready)XIC(p01r09_pb_global_reset)[OTU(p29r20.fault.2) ,OTU(p29r20.fault_ack.2) ];
   37: XIC(p29_di_wdr_turret.ready)XIO(p29_di_wdr_turret.ctrl_from_net)[TON(p29r20_timer_fault[3],?,?) ,XIC(p29r20_timer_fault[3].DN) OTL(p29r20.fault.3) ];
   38: XIC(p29r20.fault_ack.3)[XIC(p29_di_wdr_turret.ctrl_from_net) ,XIO(p29_di_wdr_turret.ready) ]XIC(p01r09_pb_global_reset)[OTU(p29r20.fault.3) ,OTU(p29r20.fault_ack.3) ];
   39: XIO(p29_di_wt_motor)[TON(p29r20_timer_fault[4],?,?) ,XIC(p29r20_timer_fault[4].DN) OTL(p29r20.fault.4) ];
   40: XIC(p29r20.fault_ack.4)XIC(p29_di_wt_motor)XIC(p01r09_pb_global_reset)[OTU(p29r20.fault.4) ,OTU(p29r20.fault_ack.4) ];
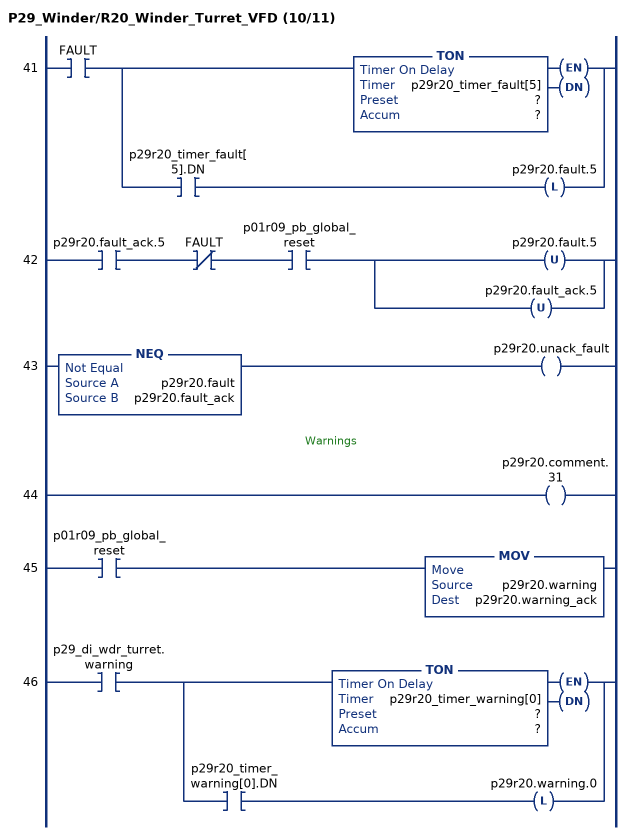
   41: XIC(FAULT)[TON(p29r20_timer_fault[5],?,?) ,XIC(p29r20_timer_fault[5].DN) OTL(p29r20.fault.5) ];
   42: XIC(p29r20.fault_ack.5)XIO(FAULT)XIC(p01r09_pb_global_reset)[OTU(p29r20.fault.5) ,OTU(p29r20.fault_ack.5) ];
   43: NEQ(p29r20.fault,p29r20.fault_ack)OTE(p29r20.unack_fault);
   // Warnings
   44: OTE(p29r20.comment.31);
   45: XIC(p01r09_pb_global_reset)MOV(p29r20.warning,p29r20.warning_ack);
   46: XIC(p29_di_wdr_turret.warning)[TON(p29r20_timer_warning[0],?,?) ,XIC(p29r20_timer_warning[0].DN) OTL(p29r20.warning.0) ];
